TYPE DUT_GetSettingRepositoryByName:
STRUCT  
	Name		: STRING(50);
	Data		: STRING(DB.MAX_STRING_SIZE);
END_STRUCT
END_TYPE

(* stored: Version 1.1.0.1, ProductVersion 3.1.4024.15
   DUT DUT_GetSettingRepositoryByName: Id {ab5b1964-9626-491c-8e52-579ae5a93535} *)
